INTERFACE IChar EXTENDS IObject

PROPERTY charAsByte : Byte
GET
END_GET
END_PROPERTY

PROPERTY charAsString : STRING(1)
GET
END_GET
END_PROPERTY

END_INTERFACE

(* stored: Version 1.1.0.1
   Itf IChar: Id {876bc023-ccfe-405d-ad4a-28a85f8c9b09}
   Property charAsByte: Id {186704e7-3046-4fa3-9745-bbd41f13bec2}
   Get Get: Id {a05506ca-9d39-4ce9-ab8d-3e27647a9a58}
   Property charAsString: Id {64f3eeeb-5ee8-4a05-8005-c79f79819de1}
   Get Get: Id {6acc084e-fcd3-4aa8-be31-d55534fb7b54} *)
